Universal Robots PolyScope program: ad_lab_exe_9_1_108.urp

Program ad_lab_exe_9_1_108 (createdIn=3.1.17195 lastSavedIn=3.2.19293 directory=/programs installation=default robotSerialNumber=2015351391)
Calibrated DH parameters: a=[0.000352, -0.161198, -0.373486, 0.00005, 0.000049, 0]; d=[0.089268, 352.477598, -320.08558, -32.281492, 0.094939, 0.082518]; alpha=[1.570728, 0.001116, -0.003686, 1.571189, -1.570572, 0]; deltaTheta=[-0.000012, 1.181849, -1.491165, 0.309495, -0.000007, 0.000025]
BeforeStart
  open := socket_open("192.168.1.6",5000)
  current_pos := p[0,0,0,0,0,0]
  Loop While (checkContinuously=false) expression=open≟ False
    open := socket_open("192.168.1.6",5000)
Robot Program (runOnlyOnce=false motionType=MoveJ speed=1.047198 acceleration=1.396263 recalculateMotions=false)
  sendToServer :=  (valueSource=Operator message=send to server valueType=String)
  Script: socket_send_string(sendToServer)
  receiveFromServ := socket_read_ascii_float(3)
  Loop While (checkContinuously=false) expression=receiveFromServ[0]≠3
    Wait Sleep waitTime=0.3
    receiveFromServ := socket_read_ascii_float(3)
  x := receiveFromServ[1]
  y := receiveFromServ[2]
  rz := d2r(receiveFromServ[3])
  current_pos := get_actual_tcp_pose()
  MoveJ speed 60 deg/s, acceleration 80 deg/s^2 (recalculateMotions=false)
    Waypoint 路点 (Variable): variable=current_pos
  offset := p[x,y,0,0,0,rz]
  target_pos := pose_trans(current_pos,offset)
  MoveJ speed 60 deg/s, acceleration 80 deg/s^2 (recalculateMotions=false)
    Waypoint 路点 (Variable): variable=target_pos
